FUNCTION_BLOCK FB_StringBuilder
VAR
END_VAR

END_FUNCTION_BLOCK

(* stored: Version 1.1.0.1
   POU FB_StringBuilder: Id {5f4330c0-fdcf-43b1-92f5-22a7ffcee2f1}, SpecialFunc None *)
